// TIA Portal project "Grespan_CLP" (V18)

(* hardware
DEVICE "S7-1200 station_1"  S7-1200 Station
   slot 0: "Rack_0"  S7-1200 Rack  Rack  V1.0
   slot 1: "CPU"  CPU 1215C DC/DC/DC  6ES7 215-1AG40-0XB0  V4.5
   slot 2: "DIQ1"  6ES7 223-1BL32-0XB0  V2.0
   slot 3: "DIQ2"  6ES7 223-1BL32-0XB0  V2.0
   slot 4: "DIQ3"  6ES7 223-1BL32-0XB0  V2.0
   slot 5: "DIQ4"  6ES7 223-1BH32-0XB0  V2.0
*)

// ===== PLC "CPU"  CPU 1215C DC/DC/DC =====

VAR_GLOBAL   // PLC tag table "Alert"
   "iBEmerencia" AT %I16.2 : Bool;
   "oSirene" AT %Q17.1 : Bool;
END_VAR

VAR_GLOBAL   // PLC tag table "01_EL-1"
   "iEL-1" AT %I0.4 : Bool;
   "oEL-1s" AT %Q17.6 : Bool;
   "oEL-1f" AT %Q17.7 : Bool;
END_VAR

VAR_GLOBAL   // PLC tag table "02_EL-2"
   "iEL-2p" AT %I0.5 : Bool;
   "iEL-2" AT %I0.6 : Bool;
   "oEL-2p" AT %Q0.0 : Bool;
   "oEL-2" AT %Q0.1 : Bool;
END_VAR

VAR_GLOBAL   // PLC tag table "03_EL-3"
   "iEL-3" AT %I0.7 : Bool;
   "oEL-3s" AT %Q20.0 : Bool;
   "oEL-3f" AT %Q20.1 : Bool;
END_VAR

VAR_GLOBAL   // PLC tag table "04_EL-4"
   "iEL-4p" AT %I1.0 : Bool;
   "iEL-4" AT %I1.1 : Bool;
   "oEL-4p" AT %Q0.2 : Bool;
   "oEL-4" AT %Q0.3 : Bool;
END_VAR

VAR_GLOBAL   // PLC tag table "05_RD-1"
   "iRD-1" AT %I1.2 : Bool;
   "oRD-1" AT %Q0.4 : Bool;
END_VAR

VAR_GLOBAL   // PLC tag table "06_RD-2"
   "iRD-2" AT %I1.3 : Bool;
   "oRD-2" AT %Q0.5 : Bool;
END_VAR

VAR_GLOBAL   // PLC tag table "07_CT-1"
   "iCT-1" AT %I1.4 : Bool;
   "oCT-1s" AT %Q20.2 : Bool;
   "oCT-1f" AT %Q20.3 : Bool;
END_VAR

VAR_GLOBAL   // PLC tag table "08_CT-2"
   "iCT-2" AT %I1.5 : Bool;
   "oCT-2s" AT %Q20.4 : Bool;
   "oCT-2f" AT %Q20.5 : Bool;
END_VAR

VAR_GLOBAL   // PLC tag table "09_CT-3"
   "iCT-3" AT %I8.0 : Bool;
   "oCT-3s" AT %Q20.6 : Bool;
   "oCT-3f" AT %Q20.7 : Bool;
END_VAR

VAR_GLOBAL   // PLC tag table "10_CT-4"
   "iCT-4p" AT %I8.1 : Bool;
   "iCT-4" AT %I8.2 : Bool;
   "oCT-4p" AT %Q0.6 : Bool;
   "oCT-4" AT %Q0.7 : Bool;
END_VAR

VAR_GLOBAL   // PLC tag table "11_CT-5"
   "iCT-5" AT %I8.3 : Bool;
   "oCT-5" AT %Q1.0 : Bool;
END_VAR

VAR_GLOBAL   // PLC tag table "12_PL-1"
   "iPL-1" AT %I8.4 : Bool;
   "oPL-1" AT %Q1.1 : Bool;
END_VAR

VAR_GLOBAL   // PLC tag table "13_SC1-EXA"
   "iSC1-EXAp" AT %I8.5 : Bool;
   "iSC1-EXA" AT %I8.6 : Bool;
   "oSC1-EXAp" AT %Q8.0 : Bool;
   "oSC1-EXA" AT %Q8.1 : Bool;
END_VAR

VAR_GLOBAL   // PLC tag table "14_SC1-ECL"
   "iSC1-ECL" AT %I8.7 : Bool;
   "oSC1-ECL" AT %Q8.2 : Bool;
END_VAR

VAR_GLOBAL   // PLC tag table "15_AE1-SA1"
   "iAE1-SA1p" AT %I9.0 : Bool;   // 3
   "iAE1-SA1" AT %I9.1 : Bool;   // 3
   "iAE1-SA1a" AT %I17.2 : Bool;
   "oAE1-SA1p" AT %Q8.3 : Bool;
   "oAE1-SA1" AT %Q8.4 : Bool;
END_VAR

VAR_GLOBAL   // PLC tag table "16_AE2-SA1"
   "iAE2-SA1p" AT %I9.2 : Bool;   // 6
   "iAE2-SA1" AT %I9.3 : Bool;   // 6
   "iAE2-SA1a" AT %I17.3 : Bool;
   "oAE2-SA1p" AT %Q8.5 : Bool;
   "oAE2-SA1" AT %Q8.6 : Bool;
END_VAR

VAR_GLOBAL   // PLC tag table "17_AE1-SA2"
   "iAE1-SA2p" AT %I9.4 : Bool;   // 4
   "iAE1-SA2" AT %I9.5 : Bool;   // 4
   "iAE1-SA2a" AT %I17.4 : Bool;
   "oAE1-SA2p" AT %Q8.7 : Bool;
   "oAE1-SA2" AT %Q9.0 : Bool;
END_VAR

VAR_GLOBAL   // PLC tag table "18_AE2-SA2"
   "iAE2-SA2p" AT %I9.6 : Bool;   // 7
   "iAE2-SA2" AT %I9.7 : Bool;   // 7
   "iAE2-SA2a" AT %I17.5 : Bool;
   "oAE2-SA2p" AT %Q9.1 : Bool;
   "oAE2-SA2" AT %Q9.2 : Bool;
END_VAR

VAR_GLOBAL   // PLC tag table "19_AE1-SA3"
   "iAE1-SA3p" AT %I12.0 : Bool;   // 5
   "iAE1-SA3" AT %I12.1 : Bool;   // 5
   "iAE1-SA3a" AT %I17.6 : Bool;
   "oAE1-SA3p" AT %Q9.3 : Bool;
   "oAE1-SA3" AT %Q9.4 : Bool;
END_VAR

VAR_GLOBAL   // PLC tag table "20_AE2-SA3"
   "iAE2-SA3p" AT %I12.2 : Bool;   // 8
   "iAE2-SA3" AT %I12.3 : Bool;   // 8
   "iAE2-SA3a" AT %I17.7 : Bool;
   "oAE2-SA3p" AT %Q9.5 : Bool;
   "oAE2-SA3" AT %Q9.6 : Bool;
END_VAR

VAR_GLOBAL   // PLC tag table "21_AER-SP1"
   "iAER-SP1p" AT %I12.4 : Bool;   // 1
   "iAER-SP1" AT %I12.5 : Bool;   // 1
   "iAER-SP1a" AT %I20.0 : Bool;
   "oAER-SP1p" AT %Q9.7 : Bool;
   "oAER-SP1" AT %Q12.0 : Bool;
END_VAR

VAR_GLOBAL   // PLC tag table "22_AER-SP2"
   "iAER-SP2p" AT %I12.6 : Bool;   // 2
   "iAER-SP2" AT %I12.7 : Bool;   // 2
   "iAER-SP2a" AT %I20.1 : Bool;
   "oAER-SP2p" AT %Q12.1 : Bool;
   "oAER-SP2" AT %Q12.2 : Bool;
END_VAR

VAR_GLOBAL   // PLC tag table "23_ESP-EG1"
   "iESP-EG1" AT %I13.0 : Bool;
   "oESP-EG1" AT %Q12.3 : Bool;
END_VAR

VAR_GLOBAL   // PLC tag table "24_ESP-EG2"
   "iESP-EG2" AT %I13.1 : Bool;
   "oESP-EG2" AT %Q12.4 : Bool;
END_VAR

VAR_GLOBAL   // PLC tag table "25_ESP-EG3"
   "iESP-EG3" AT %I13.2 : Bool;
   "oESP-EG3" AT %Q12.5 : Bool;
END_VAR

VAR_GLOBAL   // PLC tag table "26_ELR-1"
   "iELR-1" AT %I13.3 : Bool;
   "oELR-1" AT %Q12.6 : Bool;
END_VAR

VAR_GLOBAL   // PLC tag table "27_ELR-2"
   "iELR-2" AT %I13.4 : Bool;
   "oELR-2" AT %Q12.7 : Bool;
END_VAR

VAR_GLOBAL   // PLC tag table "28_ELR-3"
   "iELR-3" AT %I13.5 : Bool;
   "oELR-3" AT %Q13.0 : Bool;
END_VAR

VAR_GLOBAL   // PLC tag table "29_TOR-1"
   "iTOR-1" AT %I13.6 : Bool;
   "oTOR-1" AT %Q13.1 : Bool;
END_VAR

VAR_GLOBAL   // PLC tag table "30_EXA-1"
   "iEXA-1" AT %I13.7 : Bool;
   "oEXA-1" AT %Q13.2 : Bool;
END_VAR

VAR_GLOBAL   // PLC tag table "31_BAT-1"
   "iBAT-1" AT %I16.0 : Bool;
   "oBAT-1" AT %Q13.3 : Bool;
END_VAR

VAR_GLOBAL   // PLC tag table "32_SLR-1"
   "iSLR-1" AT %I16.1 : Bool;
   "oSLR-1" AT %Q13.4 : Bool;
END_VAR

VAR_GLOBAL   // PLC tag table "Type"
   "iSSP1p" AT %I0.0 : Bool;
   "iSSP1" AT %I0.1 : Bool;
   "iSSP2p" AT %I0.2 : Bool;
   "iSSP2" AT %I0.3 : Bool;
   "oSSP1t1" AT %Q17.2 : Bool;
   "oSSP1t2" AT %Q17.3 : Bool;
   "oSSP2t1" AT %Q17.4 : Bool;
   "oSSP2t2" AT %Q17.5 : Bool;
END_VAR

VAR_GLOBAL   // PLC tag table "Level"
   "iSP1" AT %I16.3 : Bool;
   "iSP2" AT %I16.4 : Bool;
   "iSA1" AT %I16.5 : Bool;
   "iSA2" AT %I16.6 : Bool;
   "iSA3" AT %I16.7 : Bool;
   "iTM1a" AT %I17.0 : Bool;
   "iTM1b" AT %I17.1 : Bool;
END_VAR

DATA_BLOCK "ext"   // DB1
{ S7_Optimized_Access := 'FALSE' }
VERSION : 0.1
   VAR
      block : Bool := true;
      trig : USInt;
      selector : Array[1..32] of Bool;
      status : Array[1..32] of USInt;
   END_VAR
BEGIN
   selector[15] := true;
   selector[16] := true;
   selector[17] := true;
   selector[18] := true;
   selector[19] := true;
   selector[20] := true;
   selector[21] := true;
   selector[22] := true;
   selector[1] := true;
   selector[7] := true;
   selector[3] := true;
   selector[9] := true;
   selector[8] := true;
END_DATA_BLOCK

DATA_BLOCK "int"   // DB2
{ S7_Optimized_Access := 'TRUE' }
VERSION : 0.1
   VAR
      pulse : Array[1..40] of Bool;
      tmp : Array[1..32] of IEC_TIMER;
   END_VAR
BEGIN
END_DATA_BLOCK

DATA_BLOCK "ret"   // DB3
{ S7_Optimized_Access := 'FALSE' }
VERSION : 0.1
   VAR
      switch : Array[1..17] of Bool;
   END_VAR
BEGIN
END_DATA_BLOCK

FUNCTION "fc" : Void   // FC1, SCL
{ S7_Optimized_Access := 'TRUE' }
VERSION : 0.1
   VAR_TEMP
      aux : USInt;
      null : Bool;
   END_VAR
BEGIN
   IF NOT "iBEmerencia" THEN
       #aux := "ext".trig := 0;
       FOR #aux := 1 TO 32 DO
           "ext".status[#aux] := 0;
       END_FOR;
   ELSE
       IF "ext".trig >= 1 AND "ext".trig <= 32 THEN
           IF "ext".trig >= 15 AND "ext".trig <= 22 AND "ext".selector["ext".trig] THEN
               "ext".trig := 0;
           ELSE
               IF "ext".status["ext".trig] > 0 THEN
                   "ext".status["ext".trig] := 0;
               ELSE
                   IF NOT "ext".block THEN
                       "ext".status["ext".trig] += 1;
                   ELSE
                       CASE "ext".trig OF
                           1:
                               IF NOT "ret".switch[1]  THEN //chave para cima
                                   "ext".status["ext".trig] := 1;
                               ELSE //chave para baixo
                                   IF "ext".status[7] = 1 THEN //CT-1
                                       "ext".status["ext".trig] := 1;
                                   ELSE
                                       "ext".trig := 0;
                                   END_IF;
                               END_IF;
                           2:
                               IF NOT "ret".switch[4] THEN //chave para cima
                                   "ext".status["ext".trig] := 1;
                               ELSE //chave para baixo
                                   IF "ext".status[5] = 1 THEN //RD-1
                                       "ext".status["ext".trig] := 1;
                                   ELSE
                                       "ext".trig := 0;
                                   END_IF;
                               END_IF;
                           3:
                               IF NOT "ret".switch[10] THEN //chave para cima
                                   IF NOT "ret".switch[11] THEN //chave para cima
                                       IF "ext".status[5] = 1 THEN //RD-1
                                           "ext".status["ext".trig] := 1;
                                       ELSE
                                           "ext".trig := 0;
                                       END_IF;
                                   ELSE //chave para baixo
                                       IF NOT "ret".switch[12] THEN //chave para cima
                                           IF NOT "iSP1" THEN //SP-1
                                               "ext".status["ext".trig] := 1;
                                           ELSE
                                               "ext".trig := 0;
                                           END_IF;
                                       ELSE //chave para baixo
                                           IF NOT "iSP2" THEN //SP-2
                                               "ext".status["ext".trig] := 1;
                                           ELSE
                                               "ext".trig := 0;
                                           END_IF;
                                       END_IF;
                                   END_IF;
                               ELSE //chave para baixo
                                   IF NOT "ret".switch[15] THEN //chave para cima
                                       IF "ext".status[10] = 1 THEN //CT-4
                                           "ext".status["ext".trig] := 1;
                                       ELSE
                                           "ext".trig := 0;
                                       END_IF;
                                   ELSE //chave para baixo
                                       IF NOT ("iTM1a" AND "iTM1b") THEN //TM1
                                           "ext".status["ext".trig] := 1;
                                       ELSE
                                           "ext".trig := 0;
                                       END_IF;
                                   END_IF;
                               END_IF;
                           4:
                               IF "ret".switch[16] THEN //chave para cima
                                   IF "ret".switch[14] THEN //chave para cima
                                       IF "ext".status[10] = 1 THEN //CT-4
                                           "ext".status["ext".trig] := 1;
                                       ELSE
                                           "ext".trig := 0;
                                       END_IF;
                                   ELSE //chave para baixo
                                       IF "ext".status[12] = 1 THEN //PL-1
                                           "ext".status["ext".trig] := 1;
                                       ELSE
                                           "ext".trig := 0;
                                       END_IF;
                                   END_IF;
                               ELSE //chave para baixo
                                   IF NOT ("iTM1a" AND "iTM1b") THEN //TM1
                                       "ext".status["ext".trig] := 1;
                                   ELSE
                                       "ext".trig := 0;
                                   END_IF;
                               END_IF;
                           5:
                               IF "ext".status[13] = 1 THEN //SC1-EXA
                                   "ext".status["ext".trig] := 1;
                               ELSE
                                   "ext".trig := 0;
                               END_IF;
                           6:
                               IF NOT "ret".switch[5] THEN //chave para cima
                                   IF "ext".status[2] = 1 THEN //EL-2
                                       "ext".status["ext".trig] := 1;
                                   ELSE
                                       "ext".trig := 0;
                                   END_IF;
                               ELSE //chave para baixo
                                   IF "ext".status[3] = 1 THEN //EL-3
                                       "ext".status["ext".trig] := 1;
                                   ELSE
                                       "ext".trig := 0;
                                   END_IF;
                               END_IF;
                           7:
                               IF NOT "ret".switch[2] THEN //chave para cima
                                   IF NOT "ret".switch[3] THEN //chave para cima
                                       IF "ext".status[2] = 1 THEN //EL-2
                                           "ext".status["ext".trig] := 1;
                                       ELSE
                                           "ext".trig := 0;
                                       END_IF;
                                   ELSE //chave para baixo
                                       IF "ext".status[12] = 1 THEN //PL-1
                                           "ext".status["ext".trig] := 1;
                                       ELSE
                                           "ext".trig := 0;
                                       END_IF;
                                   END_IF;
                               ELSE //chave para baixo
                                   IF NOT "ret".switch[6] THEN //chave para cima
                                       IF "ext".status[3] = 1 THEN //EL-3
                                           "ext".status["ext".trig] := 1;
                                       ELSE
                                           "ext".trig := 0;
                                       END_IF;
                                   ELSE //chave para baixo
                                       IF "ext".status[4] = 1 THEN //EL-4
                                           "ext".status["ext".trig] := 1;
                                       ELSE
                                           "ext".trig := 0;
                                       END_IF;
                                   END_IF;
                               END_IF;
                           8:
                               IF "ret".switch[8] THEN //chave para cima
                                   IF "ext".status[2] = 1 THEN //EL-2
                                       "ext".status["ext".trig] := 1;
                                   ELSE
                                       "ext".trig := 0;
                                   END_IF;
                               ELSE //chave para baixo
                                   IF "ext".status[3] = 1 THEN //EL-3
                                       "ext".status["ext".trig] := 1;
                                   ELSE
                                       "ext".trig := 0;
                                   END_IF;
                               END_IF;
                           9:
                               IF "ret".switch[13] THEN //chave para cima
                                   IF "ext".status[2] = 1 THEN //EL-2
                                       "ext".status["ext".trig] := 1;
                                   ELSE //chave para baixo
                                       "ext".trig := 0;
                                   END_IF;
                               ELSE //chave para baixo
                                   IF "ext".status[3] = 1 THEN //EL-3
                                       "ext".status["ext".trig] := 1;
                                   ELSE
                                       "ext".trig := 0;
                                   END_IF;
                               END_IF;
                           10:
                               IF "ext".status[23] = 1 OR
                                   "ext".status[24] = 1 OR
                                   "ext".status[24] = 1
                               THEN //ESP1..3
                                   "ext".status["ext".trig] := 1;
                               ELSE
                                   "ext".trig := 0;
                               END_IF;
                           11:
                               IF "ret".switch[17] THEN //chave para cima
                                   IF "ext".status[3] = 1 THEN //EL-3
                                       "ext".status["ext".trig] := 1;
                                   ELSE
                                       "ext".trig := 0;
                                   END_IF;
                               ELSE //chave para baixo
                                   IF "ext".status[4] = 1 THEN //EL-4
                                       "ext".status["ext".trig] := 1;
                                   ELSE
                                       "ext".trig := 0;
                                   END_IF;
                               END_IF;
                           12:
                               IF "ext".status[26] = 1 AND
                                   "ext".status[27] = 1 THEN //ELR1e2
                                   IF "ret".switch[7] THEN //chave para cima
                                       IF "ext".status[2] = 1 THEN //EL-2
                                           "ext".status["ext".trig] := 1;
                                       ELSE //chave para baixo
                                           "ext".trig := 0;
                                       END_IF;
                                   ELSE //chave para baixo
                                       IF "ret".switch[9] THEN //chave para cima
                                           IF "ext".status[3] = 1 THEN //EL-3
                                               "ext".status["ext".trig] := 1;
                                           ELSE
                                               "ext".trig := 0;
                                           END_IF;
                                       ELSE //chave para baixo
                                           IF "ext".status[4] = 1 THEN //EL-4
                                               "ext".status["ext".trig] := 1;
                                           ELSE
                                               "ext".trig := 0;
                                           END_IF;
                                       END_IF;
                                   END_IF;
                               ELSE //chave para baixo
                                   "ext".trig := 0;
                               END_IF;
                           13:
                               IF "ext".status[14] = 1 THEN //SC1-ECL
                                   "ext".status["ext".trig] := 1;
                               ELSE
                                   "ext".trig := 0;
                               END_IF;
                           14:
                               IF "ext".status[6] = 1 THEN //RD-2
                                   "ext".status["ext".trig] := 1;
                               ELSE
                                   "ext".trig := 0;
                               END_IF;
                           23:
                               IF "iSA1" THEN //SA-1
                                   "ext".status["ext".trig] := 1;
                               ELSE
                                   "ext".trig := 0;
                               END_IF;
                           24:
                               IF "iSA2" THEN //SA-2
                                   "ext".status["ext".trig] := 1;
                               ELSE
                                   "ext".trig := 0;
                               END_IF;
                           25:
                               IF "iSA3" THEN //SA-3
                                   "ext".status["ext".trig] := 1;
                               ELSE
                                   "ext".trig := 0;
                               END_IF;
                           27:
                               IF "ext".status[31] = 1 THEN //BAT-1
                                   "ext".status["ext".trig] := 1;
                               ELSE
                                   "ext".trig := 0;
                               END_IF;
                           28:
                               IF "ext".status[32] = 1 THEN //SLR-1
                                   "ext".status["ext".trig] := 1;
                               ELSE
                                   "ext".trig := 0;
                               END_IF;
                           29:
                               IF "ext".status[28] = 1 THEN //ELR-3
                                   "ext".status["ext".trig] := 1;
                               ELSE
                                   "ext".trig := 0;
                               END_IF;
                           32:
                               IF "ext".status[4] = 1 THEN //EL-4
                                   "ext".status["ext".trig] := 1;
                               ELSE
                                   "ext".trig := 0;
                               END_IF;
                           ELSE
                               "ext".status["ext".trig] := 1;
                       END_CASE;
                   END_IF;
               END_IF;
           END_IF;
       ELSIF "ext".trig > 0 THEN
           "ext".trig := 0;
       END_IF;
       "ext".trig := 0;
   END_IF;

   REGION Starters
       "sf" //01_EL-1 (inversor)
       (
           id          := 1,
           prm         := 2,
           inputAM     := false,
           inputSoftP  := false,
           inputP      := false,
           inputSoft   := false,
           input       := "iEL-1",
           outputP     := "oEL-1s",
           output      := "oEL-1f"
       );

       "sf" //02_EL-2 (Soft 1 Tipo 1)
       (
           id          := 2,
           prm         := 3,
           inputAM     := false,
           inputSoftP  := "iSSP1p",
           inputP      := "iEL-2p",
           inputSoft   := "iSSP1",
           input       := "iEL-2",
           outputP     := "oEL-2p",
           output      := "oEL-2"
       );

       "sf" //03_EL-3 (inversor)
       (
           id          := 3,
           prm         := 2,
           inputAM     := false,
           inputSoftP  := false,
           inputP      := false,
           inputSoft   := false,
           input       := "iEL-3",
           outputP     := "oEL-3s",
           output      := "oEL-3f"
       );

       "sf" //04_EL-4 (Soft 1 Tipo 1)
       (
           id          := 4,
           prm         := 3,
           inputAM     := false,
           inputSoftP  := "iSSP1p",
           inputP      := "iEL-4p",
           inputSoft   := "iSSP1",
           input       := "iEL-4",
           outputP     := "oEL-4p",
           output      := "oEL-4"
       );

       "sf" //05_RD-1 (Comum)
       (
           id          := 5,
           prm         := 1,
           inputAM     := false,
           inputSoftP  := false,
           inputP      := false,
           inputSoft   := false,
           input       := "iRD-1",
           outputP     := #null,
           output      := "oRD-1"
       );

       "sf" //06_RD-2 (Comum)
       (
           id          := 6,
           prm         := 1,
           inputAM     := false,
           inputSoftP  := false,
           inputP      := false,
           inputSoft   := false,
           input       := "iRD-2",
           outputP     := #null,
           output      := "oRD-2"
       );

       "sf" //07_CT-1 (inversor)
       (
           id          := 7,
           prm         := 2,
           inputAM     := false,
           inputSoftP  := false,
           inputP      := false,
           inputSoft   := false,
           input       := "iCT-1",
           outputP     := "oCT-1s",
           output      := "oCT-1f"
       );

       "sf" //08_CT-2 (inversor)
       (
           id          := 8,
           prm         := 2,
           inputAM     := false,
           inputSoftP  := false,
           inputP      := false,
           inputSoft   := false,
           input       := "iCT-2",
           outputP     := "oCT-2s",
           output      := "oCT-2f"
       );

       "sf" //09_CT-3 (inversor)
       (
           id          := 9,
           prm         := 2,
           inputAM     := false,
           inputSoftP  := false,
           inputP      := false,
           inputSoft   := false,
           input       := "iCT-3",
           outputP     := "oCT-3s",
           output      := "oCT-3f"
       );

       "sf" //10_CT-4 (Soft 2 Tipo 1)
       (
           id          := 10,
           prm         := 3,
           inputAM     := false,
           inputSoftP  := "iSSP2p",
           inputP      := "iCT-4p",
           inputSoft   := "iSSP2",
           input       := "iCT-4",
           outputP     := "oCT-4p",
           output      := "oCT-4"
       );

       "sf" //11_CT-5 (Comum)
       (
           id          := 11,
           prm         := 1,
           inputAM     := false,
           inputSoftP  := false,
           inputP      := false,
           inputSoft   := false,
           input       := "iCT-5",
           outputP     := #null,
           output      := "oCT-5"
       );

       "sf" //12_PL-1 (Comum)
       (
           id          := 12,
           prm         := 1,
           inputAM     := false,
           inputSoftP  := false,
           inputP      := false,
           inputSoft   := false,
           input       := "iPL-1",
           outputP     := #null,
           output      := "oPL-1"
       );

       "sf" //13_SC1-EXA (Soft 1 Tipo 2)
       (
           id          := 13,
           prm         := 3,
           inputAM     := false,
           inputSoftP  := "iSSP1p",
           inputP      := "iSC1-EXAp",
           inputSoft   := "iSSP1",
           input       := "iSC1-EXA",
           outputP     := "oSC1-EXAp",
           output      := "oSC1-EXA"
       );

       "sf" //14_SC1-ECL (Comum)
       (
           id          := 14,
           prm         := 1,
           inputAM     := false,
           inputSoftP  := false,
           inputP      := false,
           inputSoft   := false,
           input       := "iSC1-ECL",
           outputP     := #null,
           output      := "oSC1-ECL"
       );

       "sf" //15_AE1-SA1 (Soft 2 Tipo 2) (Auto.)
       (
           id          := 15,
           prm         := 3,
           inputAM     := "iAE1-SA1a",
           inputSoftP  := "iSSP2p",
           inputP      := "iAE1-SA1p",
           inputSoft   := "iSSP2",
           input       := "iAE1-SA1",
           outputP     := "oAE1-SA1p",
           output      := "oAE1-SA1"
       );

       "sf" //16_AE2-SA1 (Soft 1 Tipo 2) (Auto.)
       (
           id          := 16,
           prm         := 3,
           inputAM     := "iAE2-SA1a",
           inputSoftP  := "iSSP1p",
           inputP      := "iAE2-SA1p",
           inputSoft   := "iSSP1",
           input       := "iAE2-SA1",
           outputP     := "oAE2-SA1p",
           output      := "oAE2-SA1"
       );

       "sf" //17_AE1-SA2 (Soft 2 Tipo 2) (Auto.)
       (
           id          := 17,
           prm         := 3,
           inputAM     := "iAE1-SA2a",
           inputSoftP  := "iSSP2p",
           inputP      := "iAE1-SA2p"  ,
           inputSoft   := "iSSP2",
           input       := "iAE1-SA2",
           outputP     := "oAE1-SA2p",
           output      := "oAE1-SA2"
       );

       "sf" //18_AE2-SA2 (Soft 1 Tipo 2) (Auto.)
       (
           id          := 18,
           prm         := 3,
           inputAM     := "iAE2-SA2a",
           inputSoftP  := "iSSP1p",
           inputP      := "iAE2-SA2p",
           inputSoft   := "iSSP1",
           input       := "iAE2-SA2",
           outputP     := "oAE2-SA2p",
           output      := "oAE2-SA2"
       );

       "sf" //19_AE1-SA3 (Soft 2 Tipo 2) (Auto.)
       (
           id          := 19,
           prm         := 3,
           inputAM     := "iAE1-SA3a",
           inputSoftP  := "iSSP2p",
           inputP      := "iAE1-SA3p",
           inputSoft   := "iSSP2",
           input       := "iAE1-SA3",
           outputP     := "oAE1-SA3p",
           output      := "oAE1-SA3"
       );

       "sf" //20_AE2-SA3 (Soft 1 Tipo 2) (Auto.)
       (
           id          := 20,
           prm         := 3,
           inputAM     := "iAE2-SA3a",
           inputSoftP  := "iSSP1p",
           inputP      := "iAE2-SA3p",
           inputSoft   := "iSSP1",
           input       := "iAE2-SA3",
           outputP     := "oAE2-SA3p",
           output      := "oAE2-SA3"
       );

       "sf" //21_AER-SP1 (Soft 2 Tipo 2) (Auto.)
       (
           id          := 21,
           prm         := 3,
           inputAM     := "iAER-SP1a",
           inputSoftP  := "iSSP2p",
           inputP      := "iAER-SP1p",
           inputSoft   := "iSSP2",
           input       := "iAER-SP1",
           outputP     := "oAER-SP1p",
           output      := "oAER-SP1"
       );

       "sf" //22_AER-SP2 (Soft 2 Tipo 2) (Auto.)
       (
           id          := 22,
           prm         := 3,
           inputAM     := "iAER-SP2a",
           inputSoftP  := "iSSP2p",
           inputP      := "iAER-SP2p",
           inputSoft   := "iSSP2",
           input       := "iAER-SP2",
           outputP     := "oAER-SP2p",
           output      := "oAER-SP2"
       );

       "sf" //23_ESP-EG1 (Comum)
       (
           id          := 23,
           prm         := 1,
           inputAM     := false,
           inputSoftP  := false,
           inputP      := false,
           inputSoft   := false,
           input       := "iESP-EG1",
           outputP     := #null,
           output      := "oESP-EG1"
       );

       "sf" //24_ESP-EG2 (Comum)
       (
           id          := 24,
           prm         := 1,
           inputAM     := false,
           inputSoftP  := false,
           inputP      := false,
           inputSoft   := false,
           input       := "iESP-EG2",
           outputP     := #null,
           output      := "oESP-EG2"
       );

       "sf" //25_ESP-EG3 (Comum)
       (
           id          := 25,
           prm         := 1,
           inputAM     := false,
           inputSoftP  := false,
           inputP      := false,
           inputSoft   := false,
           input       := "iESP-EG3",
           outputP     := #null,
           output      := "oESP-EG3"
       );

       "sf" //26_ELR-1 (Comum)
       (
           id          := 26,
           prm         := 1,
           inputAM     := false,
           inputSoftP  := false,
           inputP      := false,
           inputSoft   := false,
           input       := "iELR-1",
           outputP     := #null,
           output      := "oELR-2"
       );

       "sf" //27_ELR-2 (Comum)
       (
           id          := 27,
           prm         := 1,
           inputAM     := false,
           inputSoftP  := false,
           inputP      := false,
           inputSoft   := false,
           input       := "iELR-2",
           outputP     := #null,
           output      := "oELR-2"
       );

       "sf" //28_ELR-3 (Comum)
       (
           id          := 28,
           prm         := 1,
           inputAM     := false,
           inputSoftP  := false,
           inputP      := false,
           inputSoft   := false,
           input       := "iELR-3",
           outputP     := #null,
           output      := "oELR-3"
       );

       "sf" //29_TOR-1 (Comum)
       (
           id          := 29,
           prm         := 1,
           inputAM     := false,
           inputSoftP  := false,
           inputP      := false,
           inputSoft   := false,
           input       := "iTOR-1",
           outputP     := #null,
           output      := "oTOR-1"
       );

       "sf" //30_EXA-1 (Comum)
       (
           id          := 30,
           prm         := 1,
           inputAM     := false,
           inputSoftP  := false,
           inputP      := false,
           inputSoft   := false,
           input       := "iEXA-1",
           outputP     := #null,
           output      := "oEXA-1"
       );

       "sf" //31_BAT-1 (Comum)
       (
           id          := 31,
           prm         := 1,
           inputAM     := false,
           inputSoftP  := false,
           inputP      := false,
           inputSoft   := false,
           input       := "iBAT-1",
           outputP     := #null,
           output      := "oBAT-1"
       );

       "sf" //32_SLR-1 (Comum)
       (
           id          := 32,
           prm         := 1,
           inputAM     := false,
           inputSoftP  := false,
           inputP      := false,
           inputSoft   := false,
           input       := "iSLR-1",
           outputP     := #null,
           output      := "oSLR-1"
       );

       REGION Soft Type

           IF "oEL-2p" OR "oEL-4p" THEN
               "oSSP1t1" := true;
           ELSE
               "oSSP1t1" := false;
           END_IF;

           IF "oSC1-EXAp" OR "oAE2-SA1p" OR "oAE2-SA2p" OR "oAE2-SA3p" THEN
               "oSSP1t2" := true;
           ELSE
               "oSSP1t2" := false;
           END_IF;

           IF "oCT-4p" THEN
               "oSSP2t1" := true;
           ELSE
               "oSSP2t1" := false;
           END_IF;

           IF "oAE1-SA1p" OR "oAE1-SA2p" OR "oAE1-SA3p" OR "oAER-SP1p" OR "oAER-SP2p" THEN
               "oSSP2t2" := true;
           ELSE
               "oSSP2t2" := false;
           END_IF;
       END_REGION

   END_REGION

   #aux := 0;
   FOR #aux := 1 TO 40 DO
       IF "int".pulse[#aux] THEN
           "oSirene" := true;
       END_IF;
   END_FOR;
END_FUNCTION

FUNCTION "sf" : Void   // FC2, SCL
{ S7_Optimized_Access := 'TRUE' }
VERSION : 0.1
   VAR_INPUT
      id : USInt;
      prm : USInt;
      inputAM : Bool;
      inputSoftP : Bool;
      inputP : Bool;
      inputSoft : Bool;
      input : Bool;
   END_VAR
   VAR_IN_OUT
      outputP : Bool;
      output : Bool;
   END_VAR
BEGIN
   "int".tmp[#id].TP
   (
       PT := T#1s,
       IN := "ext".status[#id] = 1 OR #inputSoft
   );

   CASE #prm OF
       1:  // Partida Direta
           CASE "ext".status[#id] OF
               0:
                   #output := false;
               1:
                   IF "int".tmp[#id].Q OR #input THEN
                       #output := true;
                   ELSE
                       "ext".status[#id] := 3;
                   END_IF;
               3:
                   #output := false;
               ELSE
                   "ext".status[#id] := 0;
           END_CASE;

       2:  // Partida por Inversor de frequência
           CASE "ext".status[#id] OF
               0:
                   #output := false;
               1:
                   IF "int".tmp[#id].Q OR #input THEN
                       #output := true;
                   ELSE
                       "ext".status[#id] := 3;
                   END_IF;
               3:
                   #output := false;
               ELSE
                   "ext".status[#id] := 0;
           END_CASE;
           IF NOT "ext".selector[#id] AND #output THEN
               #outputP := true;
           ELSE
               #outputP := false;
           END_IF;

       3:  // Partida por Soft Starter
           IF "ext".selector[#id] THEN
               IF #inputAM AND NOT ("ext".status[#id] = 1) THEN
                   "ext".status[#id] := 1;
               ELSIF NOT #inputAM THEN
                   "ext".status[#id] := 0;
               END_IF;
           END_IF;
           CASE "ext".status[#id] OF
               0:
                   #output := #outputP := false;
                   RESET_TIMER("int".tmp[#id]);
               1:
                   IF NOT (#inputSoft OR #output) THEN
                       IF (#inputSoftP AND NOT #outputP AND NOT #output) THEN
                           "ext".status[#id] := 0;
                       ELSIF ("int".tmp[#id].ET < T#10s AND NOT #output) OR
                           (#inputP AND #inputSoftP) THEN
                           #outputP := true;
                       ELSE
                           "ext".status[#id] := 3;
                       END_IF;
                       IF #inputP AND #inputSoftP THEN
                           RESET_TIMER("int".tmp[#id]);
                       END_IF;
                   ELSE
                       IF "int".tmp[#id].ET < T#1s OR #input THEN
                           #output := true;
                       ELSE
                           "ext".status[#id] := 3;
                       END_IF;
                       #outputP := false;
                   END_IF;

               3:
                   #output := #outputP := false;
               ELSE
                   "ext".status[#id] := 0;
           END_CASE;
   END_CASE;

   IF "ext".status[#id] = 3 AND NOT "int".pulse[#id] THEN
       "int".pulse[#id] := true;
   ELSIF NOT ("ext".status[#id] = 3) THEN
       "int".pulse[#id] := false;
   END_IF;
END_FUNCTION

ORGANIZATION_BLOCK "main"   // OB1, SCL, ProgramCycle
TITLE = "Main Program Sweep (Cycle)"
{ S7_Optimized_Access := 'TRUE' }
VERSION : 0.1
   VAR_INPUT
      Initial_Call : Bool;   // Initial call of this OB
      Remanence : Bool;   // =True, if remanent data are available
   END_VAR
BEGIN
   "fc"();
END_ORGANIZATION_BLOCK